(* CODESYS project HeatSealMotor.xml

Project tree, tasks and I/O mapping:
  function block HeatSealMotor [LD]
*)

// HeatSealMotor
FUNCTION_BLOCK HeatSealMotor
// Z2 WHITE 
// U2 RED
// U1 BLACK
// MB ORANGE
// MB ORANGE
//  .					.					.
VAR_INPUT
	Forward: 			BOOL;				//
	Reverse: 			BOOL;				//
	Brake: 				BOOL;				//
	Settings: 			MotorSettings;		//
END_VAR
VAR_OUTPUT
	MotorOutput: 		BOOL;				//
	ReverseOutput: 		BOOL;				//
	BrakeOutput: 		BOOL;				//
END_VAR
VAR
END_VAR

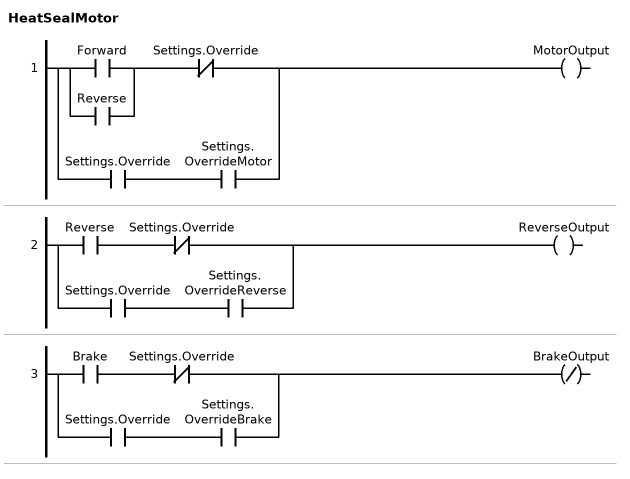
// NETWORK 1
MotorOutput := (Forward OR Reverse) AND NOT Settings.Override OR Settings.Override AND Settings.OverrideMotor;

// NETWORK 2
ReverseOutput := Reverse AND NOT Settings.Override OR Settings.Override AND Settings.OverrideReverse;

// NETWORK 3
BrakeOutput := NOT (Brake AND NOT Settings.Override OR Settings.Override AND Settings.OverrideBrake);

END_FUNCTION_BLOCK
